KUKA KRL data list: A04_swp_global.dat

&ACCESS RV
&COMMENT V_1_4_0
DEFDAT A04_swp_global PUBLIC
;********************************
;Date: 07.11.2018
;Programmer: AIUT
;Description: Global positions
;********************************



ENDDAT
